// TIA Portal project "Traffic lightss" (V16)

(* hardware
DEVICE "S7300/ET200M station_1"  S7-300 station
   slot 0: "Rail_0"  Rail  6ES7 390-1***0-0AA0
   slot 2: "PLC_1"  CPU 313C-2 DP  6ES7 313-6CF03-0AB0  V2.6
      slot 0: "MPI interface_1"  X1
      slot 1: "DP interface_1"  X2
      slot 2: "DI 16/DO 16_1"  DI16/DO16
      slot 4: "Count_1"  Counter
*)

// ===== PLC "PLC_1"  CPU 313C-2 DP =====

VAR_GLOBAL   // PLC tag table "Default tag table"
   "Red" AT %Q0.0 : Bool;
   "Green" AT %Q0.1 : Bool;
   "Yellow" AT %Q0.2 : Bool;
   "t1" AT %M0.0 : Bool;
END_VAR

ORGANIZATION_BLOCK "Main"   // OB1, LAD
TITLE = "Main Program Sweep (Cycle)"
{ S7_Optimized_Access := 'FALSE' }
VERSION : 0.1
   VAR_TEMP
      OB1_EV_CLASS : Byte;   // Bits 0-3 = 1 (Coming event), Bits 4-7 = 1 (Event class 1)
      OB1_SCAN_1 : Byte;   // 1 (Cold restart scan 1 of OB 1), 3 (Scan 2-n of OB 1)
      OB1_PRIORITY : Byte;   // Priority of OB Execution
      OB1_OB_NUMBR : Byte;   // 1 (Organization block 1, OB1)
      OB1_RESERVED_1 : Byte;   // Reserved for system
      OB1_RESERVED_2 : Byte;   // Reserved for system
      OB1_PREV_CYCLE : Int;   // Cycle time of previous OB1 scan (milliseconds)
      OB1_MIN_CYCLE : Int;   // Minimum cycle time of OB1 (milliseconds)
      OB1_MAX_CYCLE : Int;   // Maximum cycle time of OB1 (milliseconds)
      OB1_DATE_TIME : Date_And_Time;   // Date and time OB1 started
   END_VAR
   VAR_TEMP   // added for the SCL form of the ladder/FBD networks
      _w1 : Bool;
   END_VAR
BEGIN

REGION Network 1
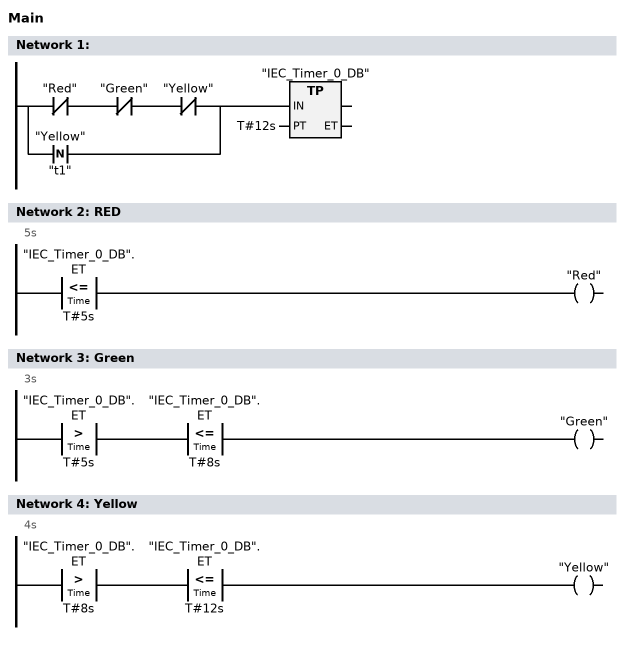
   #_w1 := NOT "Yellow" AND "t1";   // falling edge of "Yellow"
   "t1" := "Yellow";
   "IEC_Timer_0_DB".TP(IN := (NOT "Red" AND NOT "Green" AND NOT "Yellow") OR #_w1, PT := T#12s);
END_REGION

REGION Network 2: RED
   // 5s
   RUNG wire#powerrail
      { S7_Templates := "SrcType := Time" } LE_Contact(in1 := "IEC_Timer_0_DB".ET, in2 := T#5s)
      Coil( "Red" )
   END_RUNG
   // the same network as SCL:
   "Red" := "IEC_Timer_0_DB".ET <= T#5s;
END_REGION

REGION Network 3: Green
   // 3s
   RUNG wire#powerrail
      { S7_Templates := "SrcType := Time" } GT_Contact(in1 := "IEC_Timer_0_DB".ET, in2 := T#5s)
      { S7_Templates := "SrcType := Time" } LE_Contact(in1 := "IEC_Timer_0_DB".ET, in2 := T#8s)
      Coil( "Green" )
   END_RUNG
   // the same network as SCL:
   "Green" := ("IEC_Timer_0_DB".ET > T#5s) AND ("IEC_Timer_0_DB".ET <= T#8s);
END_REGION

REGION Network 4: Yellow
   // 4s
   RUNG wire#powerrail
      { S7_Templates := "SrcType := Time" } GT_Contact(in1 := "IEC_Timer_0_DB".ET, in2 := T#8s)
      { S7_Templates := "SrcType := Time" } LE_Contact(in1 := "IEC_Timer_0_DB".ET, in2 := T#12s)
      Coil( "Yellow" )
   END_RUNG
   // the same network as SCL:
   "Yellow" := ("IEC_Timer_0_DB".ET > T#8s) AND ("IEC_Timer_0_DB".ET <= T#12s);
END_REGION
END_ORGANIZATION_BLOCK